(*Created by Beckhoff*)

TYPE udt_AX5000Diag :
STRUCT
	(* NC-Status *)
	nNCAxisID				: UDINT;
	bOperational				: BOOL;
	bC1DError				: BOOL;
	bWcStateError			: BOOL;
	bAxisError				: BOOL;
	iAxisErrorCode			: UDINT;

	(* Drive Diag *)
	strDriveType				: STRING(19);
	strMotorType				:STRING(31);
	wDriveStatus				: WORD;
	wClass1Diag				: WORD;
	stClass1Diag				: ST_AX5000_C1D;
	stDriveStatus				: ST_AX5000DriveStatus;
	stEcSlaveStateBits		: ST_EcSlaveStateBits;
	stEcSlaveState			: ST_EcSlaveState;
	bPreopToSafeOpError		: BOOL;
	bSafeOpToOpError		: BOOL;
	stCPxInvParamList			:ST_SoE_CPxInvParamList;
	iDiagNumber				: UDINT;
	stDiagNumberList			:ST_SoE_DiagNumList;
	strDiagMessage			: STRING(19);
	strDiagMessageFull		: STRING(60);
END_STRUCT
END_TYPE

(* stored: Version 1.1.0.1, ProductVersion 3.1.4024.5
   DUT udt_AX5000Diag: Id {15aff478-8eaf-49a2-addc-3dcccc40ebbe} *)
